// TIA Portal V21 export
FUNCTION_BLOCK "On Delay Timer"   // FB150, LAD
{ S7_Optimized_Access := 'FALSE' }
// stored: AutoNumber false, SetENOAutomatically false
   VAR_INPUT
      TIME_START : Bool;
      TIME_PULSE : Bool;
      TIME_IN_SEC : Int;
   END_VAR
   VAR_IN_OUT
      DONE_BIT : Bool;
      ES_SEC : Int;
   END_VAR
   VAR_TEMP   // added for the SCL form of the ladder/FBD networks
      _w1 : Bool;
   END_VAR
BEGIN

REGION Network 1
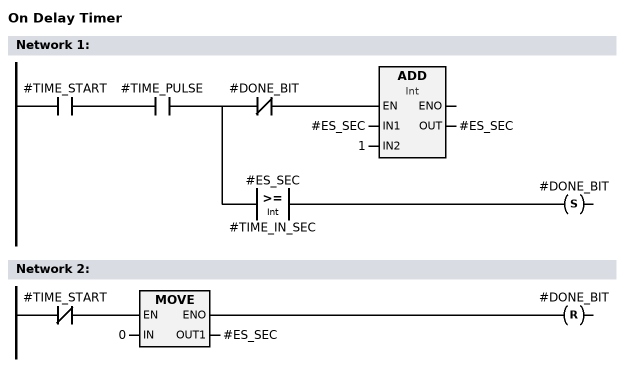
   RUNG wire#powerrail
      Contact( #TIME_START )
      Contact( #TIME_PULSE )
      wire#w1
      I_Contact( #DONE_BIT )
      { S7_Templates := "SrcType := Int"; S7_GenerateENO := "TRUE" } Add(in1 := #ES_SEC, in2 := 1, out => #ES_SEC)
   END_RUNG
   RUNG wire#w1
      { S7_Templates := "SrcType := Int" } GE_Contact(in1 := #ES_SEC, in2 := #TIME_IN_SEC)
      S_Coil( #DONE_BIT )
   END_RUNG
   // the same network as SCL:
   #_w1 := #TIME_START AND #TIME_PULSE;
   IF #_w1 AND NOT #DONE_BIT THEN #ES_SEC := #ES_SEC + 1; END_IF;
   IF #_w1 AND (#ES_SEC >= #TIME_IN_SEC) THEN #DONE_BIT := TRUE; END_IF;
END_REGION

REGION Network 2
   RUNG wire#powerrail
      I_Contact( #TIME_START )
      { S7_GenerateENO := "TRUE" } Move(in := 0, out1 => #ES_SEC)
      R_Coil( #DONE_BIT )
   END_RUNG
   // the same network as SCL:
   // ENO of a box is taken as its EN; it also drops when the box reports an error
   IF NOT #TIME_START THEN
       #ES_SEC := 0;
       #DONE_BIT := FALSE;
   END_IF;
END_REGION
END_FUNCTION_BLOCK
